FUNCTION_BLOCK T_StructFromJsonFileReader EXTENDS T_NamedBase
VAR
	filePath : STRING; // fully qualified, including directory
	fileRead : T_FileReadBase;
	jDoc : JsonDoc;
	structureName : STRING; // i.e. 'ST_Recipe'
	pointerToStructure : PVOID; // i.e. ADR(recipe)
	sizeOfStructure : UDINT; // i.e. SIZEOF(recipe) 
	jsonDataTypeWriter : FB_JsonReadWriteDataType;
	_error : BOOL;
	_busy : BOOL;
	_done : BOOL;
	_fileExists : BOOL;
	doneTrig : R_TRIG;
END_VAR

fileRead();
_error S= fileRead.Error;
_busy := fileRead.Busy;
_done := fileRead.Done AND fileRead.BufferAvailable;
_fileExists := fileRead.FileExists;

doneTrig( CLK := _done );

IF doneTrig.Q AND NOT _error THEN
	// clear jDoc
	MEMSET( ADR( jDoc ), 0, SIZEOF( jDoc ) );
	
	// get the data into the doc
	MEMCPY(
		destAddr := ADR( jDoc ),
		srcAddr := fileRead.DataBuffer,
		n := fileRead.DataLength
	);
	
	// conver the doc to the structure
	_error S= NOT jsonDataTypeWriter.SetSymbolFromJson(
		sJson := jDoc,
		sDatatype := structureName,
		nData := sizeOfStructure,
		pData := pointerToStructure
	);

END_IF

{attribute 'monitoring' := 'call' }
PROPERTY PUBLIC Busy : BOOL
GET
Busy := _busy;
END_GET
END_PROPERTY

{attribute 'monitoring' := 'call' }
PROPERTY PUBLIC Done : BOOL
GET
Done := _done;
END_GET
END_PROPERTY

{attribute 'monitoring' := 'call' }
PROPERTY PUBLIC Error : BOOL
GET
Error := _error;
END_GET
END_PROPERTY

{attribute 'monitoring' := 'call'}
PROPERTY PUBLIC FileExists : BOOL
GET
FileExists := _fileExists;
END_GET
END_PROPERTY

METHOD ReadFromFile // start the read.
IF _error THEN
	LogError ( 'Cannot read from file while block is in an error state. Reset first' );
	RETURN;
	
END_IF

_error S= NOT fileRead.StartRead();

IF _error THEN
	LogError ( 'ReadFromFile error, try Rest or wait until not busy' );
	RETURN;
	
END_IF
END_METHOD

METHOD PUBLIC Reset
_error := FALSE;
LogDebug( 'Reset called' );
END_METHOD

METHOD PUBLIC SetFileParams
VAR_INPUT
	FilePath : Tc2_Utilities.T_MaxString;
	StructureName : STRING; // i.e. 'ST_Recipe'
	PointerToStructure : PVOID; // i.e. ADR(recipe) 
	SizeOfStructure : UDINT; // i.e. SIZEOF(recipe) 
END_VAR
THIS^.filePath := FilePath; // for debug only.
fileRead.SetFilePath( FilePath := FilePath );

THIS^.structureName := StructureName;
THIS^.pointerToStructure := PointerToStructure; 
THIS^.sizeOfStructure := SizeOfStructure;
END_METHOD

END_FUNCTION_BLOCK

(* stored: Version 1.1.0.1, ProductVersion 3.1.4022.18
   POU T_StructFromJsonFileReader: Id {016623f6-0ecd-07dc-1a87-4776279e0b49}, SpecialFunc None
   Property Busy: Id {4a4da27e-b4d5-0694-0f0a-993b08e51804}
   Get Get: Id {5f53de3c-cdc2-073c-2e1d-45486d372afa}
   Property Done: Id {5399fb37-82ba-0415-11f9-314370e9e75d}
   Get Get: Id {af18cdd6-2c2a-0ab1-0613-ebf6e8dbafa2}
   Property Error: Id {ef5c5a2d-3d38-00a6-3b96-1f936bf87f33}
   Get Get: Id {0eb42b2d-cbf9-0d70-2903-f822c1680ea6}
   Property FileExists: Id {2283cf80-96f4-04bc-12ac-a182f3cd8ddd}
   Get Get: Id {3332bbdb-c463-058e-3f44-622bc70cd6a1}
   Method ReadFromFile: Id {07a81e8b-c4b9-0ac3-06f1-49b4bce3279b}
   Method Reset: Id {9526566b-fa8a-0559-3909-b287cebea629}
   Method SetFileParams: Id {4a33faa7-9971-01fa-095a-8b3bf1caabd5} *)
